# EPICS substitutions: bsaDriverApp/Db/bsa.substitutions
file bsaLinearConversion.db {
    pattern { _NOTHING_TODO_ }
            { _NOTHING_TODO_ }
}

file devScBsaHst.db {
    pattern {  INST,  MDID,   MAXLENGTH      }
#
# user Edefs
#
            {  "21",  "21",  "\$\(BSA_LENGTH=20000\)"  }
            {  "22",  "22",  "\$\(BSA_LENGTH=20000\)"  }
            {  "23",  "23",  "\$\(BSA_LENGTH=20000\)"  }
            {  "24",  "24",  "\$\(BSA_LENGTH=20000\)"  }
            {  "25",  "25",  "\$\(BSA_LENGTH=20000\)"  }
            {  "26",  "26",  "\$\(BSA_LENGTH=20000\)"  }
            {  "27",  "27",  "\$\(BSA_LENGTH=20000\)"  }
            {  "28",  "28",  "\$\(BSA_LENGTH=20000\)"  }
            {  "29",  "29",  "\$\(BSA_LENGTH=20000\)"  }
            {  "30",  "30",  "\$\(BSA_LENGTH=20000\)"  }
#
            {  "31",  "31", "\$\(BSA_LENGTH=20000\)"  }
            {  "32",  "32", "\$\(BSA_LENGTH=20000\)"  }
            {  "33",  "33", "\$\(BSA_LENGTH=20000\)"  }
            {  "34",  "34", "\$\(BSA_LENGTH=20000\)"  }
            {  "35",  "35", "\$\(BSA_LENGTH=20000\)"  }
            {  "36",  "36", "\$\(BSA_LENGTH=20000\)"  }
            {  "37",  "37", "\$\(BSA_LENGTH=20000\)"  }
            {  "38",  "38", "\$\(BSA_LENGTH=20000\)"  }
            {  "39",  "39", "\$\(BSA_LENGTH=20000\)"  }
            {  "40",  "40", "\$\(BSA_LENGTH=20000\)"  }
#
            {  "41",  "41", "\$\(BSA_LENGTH=20000\)"  }
            {  "42",  "42", "\$\(BSA_LENGTH=20000\)"  }
            {  "43",  "43", "\$\(BSA_LENGTH=20000\)"  }
            {  "44",  "44", "\$\(BSA_LENGTH=20000\)"  }
            {  "45",  "45", "\$\(BSA_LENGTH=20000\)"  }
            {  "46",  "46", "\$\(BSA_LENGTH=20000\)"  }
            {  "47",  "47", "\$\(BSA_LENGTH=20000\)"  }
            {  "48",  "48", "\$\(BSA_LENGTH=20000\)"  }
            {  "49",  "49", "\$\(BSA_LENGTH=20000\)"  }
#
# system Edefs
#
            {  "50",  "SCD1H", "\$\(BSA_LENGTH=20000\)"  }
#
            {  "51",  "SCDTH", "\$\(BSA_LENGTH=20000\)"  }
            {  "52",  "SCDHH", "\$\(BSA_LENGTH=20000\)"  }
            {  "53",  "SCL1H", "\$\(BSA_LENGTH=20000\)"  }
            {  "54",  "SCLTH", "\$\(BSA_LENGTH=20000\)"  }
            {  "55",  "SCLHH", "\$\(BSA_LENGTH=20000\)"  }
            {  "56",  "SCB1H", "\$\(BSA_LENGTH=20000\)"  }
            {  "57",  "SCBTH", "\$\(BSA_LENGTH=20000\)"  }
            {  "58",  "SCBHH", "\$\(BSA_LENGTH=20000\)"  }
            {  "59",  "SCH1H", "\$\(BSA_LENGTH=20000\)"  }
            {  "60",  "SCHTH", "\$\(BSA_LENGTH=20000\)"  }
#
            {  "61",  "SCHHH", "\$\(BSA_LENGTH=20000\)"  }
            {  "62",  "SCS1H", "\$\(BSA_LENGTH=20000\)"  }
            {  "63",  "SCSTH", "\$\(BSA_LENGTH=20000\)"  }
            {  "64",  "SCSHH", "\$\(BSA_LENGTH=20000\)"  }
#
# fault buffer
#
            {  "65",  "FLTB0", "\$\(FLTB_LENGTH=1000000\)" }
            {  "66",  "FLTB1", "\$\(FLTB_LENGTH=1000000\)" }
            {  "67",  "FLTB2", "\$\(FLTB_LENGTH=1000000\)" }
            {  "68",  "FLTB3", "\$\(FLTB_LENGTH=1000000\)" }
#
}
